{attribute 'GeneratedUsingTerminal: '}
{attribute addProperty BoxType ""}
{attribute addProperty Id "_defaultAT %I*SyncUnitTasks_D3C9946A27"}
{attribute addProperty CRC "1039812589"}
{attribute addProperty Size "27"}
TYPE SyncUnits_3DFA47ED :
STRUCT
	{attribute addProperty Name "_default"}
	_default : SyncUnitTasks_D3C9946A;
END_STRUCT
END_TYPE

(* stored: Version 1.2.0.0, ProductVersion 3.1.4024.9
   DUT SyncUnits_3DFA47ED: Id {b1d2b8e5-a38d-44fd-b88b-4605aa53c593} *)
